// TIA Portal project "MOVE" (V19)

(* hardware
DEVICE "SIMATIC 1200 station_1"  S71200.Device
   slot 0: "S7-1200 rack"  Rack  V1.0
   slot 1: "PLC_1"  CPU 1214C DC/DC/DC  6ES7 214-1AG40-0XB0  V4.0
   slot 3: "AQ1 x 12 bits_1"  6ES7 232-4HA30-0XB0  V1.0
DEVICE "HMI_1"  KTP600 Basic color PN
   slot 0: "HMI"  HMI  6AV6 647-0AD11-3AX0  12.0.0.0
   slot 1: "HMI_RT_1"  KTP600 Basic color PN  6AV6 647-0AD11-3AX0  12.0.0.0
   slot 5: "IE_CP_1"  PROFINET Interface  IE_CP  V7.1.0
      slot 1: "PROFINET_Interface_1"  PROFINET Interface
         slot 1: "PORT_1"  Port  1.0.0.0
*)

// ===== PLC "PLC_1"  CPU 1214C DC/DC/DC =====

VAR_GLOBAL   // PLC tag table "Default tag table"
   "SEL_SW_1" AT %I0.0 : Bool;   // Selector Switch, Position 1
   "SEL_SW_2" AT %I0.1 : Bool;   // Selector Switch, Position 2
   "SEL_SW_3" AT %I0.2 : Bool;   // Selector Switch, Position 3
   "START" AT %I0.4 : Bool;   // START Momentary N. O. Pushbutton
   "OUTPUT" AT %Q0.0 : Bool;   // Process Output
END_VAR

DATA_BLOCK "Data_block_Presets"   // DB1
{ S7_Optimized_Access := 'TRUE' }
VERSION : 0.1
   VAR RETAIN
      PRE_SET_1 : Int := 10000;   // Preset No. 1
      PRE_SET_2 : Int := 15000;   // Preset No. 2
      PRE_SET_3 : Int := 20000;   // Preset No. 3
   END_VAR
   VAR
      ONE_SHOT : Array[0..2] of Bool;   // One Shot Control
   END_VAR
BEGIN
END_DATA_BLOCK

// folder: System blocks/Program resources

DATA_BLOCK "DWELL"   // DB2
{ S7_Optimized_Access := 'TRUE' }
AUTHOR : Simatic
FAMILY : IEC
NAME : IEC_TMR
VERSION : 1.0
// stored: InstanceOfName IEC_TIMER
"IEC_TIMER"
BEGIN
END_DATA_BLOCK

// folder: (top level)

ORGANIZATION_BLOCK "Main"   // OB1, LAD, ProgramCycle
TITLE = "Main Program Sweep (Cycle)"
{ S7_Optimized_Access := 'TRUE' }
VERSION : 0.1
BEGIN

REGION Network 1
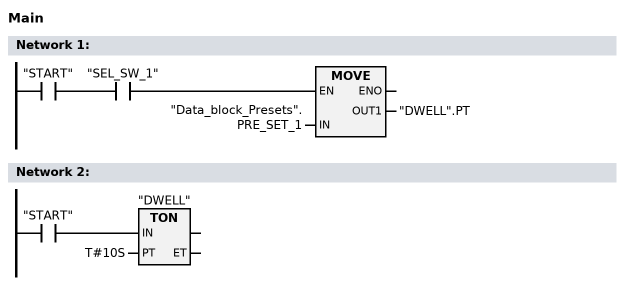
   RUNG wire#powerrail
      Contact( "START" )
      Contact( "SEL_SW_1" )
      Move(in := "Data_block_Presets".PRE_SET_1, out1 => "DWELL".PT)
   END_RUNG
   // the same network as SCL:
   IF "START" AND "SEL_SW_1" THEN "DWELL".PT := "Data_block_Presets".PRE_SET_1; END_IF;
END_REGION

REGION Network 2
   "DWELL".TON(IN := "START", PT := T#10S);
END_REGION
END_ORGANIZATION_BLOCK

(* ===== HMI "HMI_RT_1" =====
system functions are stored by id; their names below are inferred from use
connection "HMI_connection": ETHERNET, SMART_S7_1200_OMS

HMI tags "Default tag table"
   "OUTPUT" : Bool = PLC OUTPUT AT %Q0.0, 1 s
   "Data_block_HMI_OP_PB" : Int = PLC Data_block_HMI.HMI_PB, 1 s
   "Data_block_HMI_OP_START" : Bool = PLC Data_block_HMI.HMI_START, 1 s
   "Data_block_HMI_OP_PT" : Real = PLC Data_block_HMI.HMI_PT, 1 s
   "Data_block_HMI_OP_ET" : Real = PLC Data_block_HMI.HMI_ET, 1 s
   "Data_block_HMI_ENABLE_DISABLE" : Bool = PLC Data_block_HMI.HMI_ENABLE_DISABLE, 1 s
   "Data_block_Presets_PRE_SET_1" : Int = PLC Data_block_Presets.PRE_SET_1, 1 s
   "Data_block_Presets_PRE_SET_2" : Int = PLC Data_block_Presets.PRE_SET_2, 1 s
   "Data_block_Presets_PRE_SET_3" : Int = PLC Data_block_Presets.PRE_SET_3, 1 s

Template "Template_1" 320x240
   Softkey "Softkey_F6" at 266,202 size 53x38
      on KeyUp: StopRuntime(0)
   Button "Template_Button_1" at 268,202 size 51x37; TextOff 'Text'; PictureOff "ExitRuntime_HMI_1"
      on Release: StopRuntime(0)

screen "Root screen" 320x240, template "Template_1"
   GraphicView "D3_Plate_Vertical_Broad" at 13,33 size 106x165; Picture "Design_3_Plate_Vertical_Broad"
   GraphicView "D3_Plate_Vertical_Broad_1" at 128,33 size 184x164; Picture "Design_3_Plate_Vertical_Broad"
   Button "Button_1" at 47,60 size 36x36; TextOff '1'
      on Release: SetTag("Data_block_HMI_OP_PB", 1)
   TextField "Text field_1" at 25,38 size 80x18; Text 'TIME SELECT'
   Button "Button_2" at 47,104 size 36x36; TextOff '2'
      on Release: SetTag("Data_block_HMI_OP_PB", 2)
   Button "Button_3" at 47,149 size 36x36; TextOff '3'
      on Release: SetTag("Data_block_HMI_OP_PB", 3)
   IOField "I/O field_1" at 214,149 size 80x23; FormatPattern 99.99
      ProcessValue <- "Data_block_HMI_OP_ET"
   Button "Button_4" at 144,53 size 91x30; TextOff 'START'
      on Press: SetBit("Data_block_HMI_OP_START")
      on Release: ResetBit("Data_block_HMI_OP_START")
   IOField "I/O field_2" at 214,108 size 80x23; FormatPattern 99.99
      ProcessValue <- "Data_block_HMI_OP_PT"
   TextField "Text field_2" at 34,4 size 252x21; Text 'MOVE LAB OPERATORS PANEL'
   Circle "Circle_1" at 254,57 size 32x32
      Appearance <- "OUTPUT"
   TextField "Text field_4" at 140,106 size 68x15; Text 'TIME DELAY'
   TextField "Text field_5" at 150,117 size 48x16; Text 'PRESET'
   TextField "Text field_6" at 148,145 size 53x15; Text 'CURRENT'
   TextField "Text field_7" at 159,156 size 30x15; Text 'TIME'
   TextField "Text field_3" at 247,40 size 47x15; Text 'OUTPUT'
   Button "Button_5" at 1,202 size 51x37; TextOff 'SCREEN 2'
      on Release: ActivateScreen("Screen_2", 0)
   TextField "Text field_8" at 68,200 size 105x35; Text 'OVERRIDE FOR HARDWIRED OPERATOR'S PANEL'
   Switch "Switch_1" at 180,202 size 69x33; CaptionText 'Switch'; TextOff 'HMI DISABLED'; TextOn 'HMI ENABLED'
      ProcessValue <- "Data_block_HMI_ENABLE_DISABLE"
   Softkey "Softkey_F1" at 1,202 size 53x38
      on KeyUp: ActivateScreen("Screen_2", 0)

screen "Screen_2" 320x240, template "Template_1"
   Softkey "Softkey_F1" at 1,202 size 53x38
      on KeyUp: ActivateScreen("Root screen", 0)
   Button "Button_1" at 2,201 size 51x37; TextOff 'SCREEN 1'
      on Release: ActivateScreen("Root screen", 0)
   TextField "Text field_2" at 31,4 size 258x21; Text 'PRESET MAINTENANCE PANEL'
   GraphicView "D3_Plate_Vertical_Broad_1" at 59,34 size 203x163; Picture "Design_3_Plate_Vertical_Broad"
   TextField "Text field_1" at 81,41 size 160x28; Text 'ENTER VALUES AS INTEGERS TIMEBASE OF MILLISECONDS'
   TextField "Text field_3" at 82,77 size 60x18; Text 'PRESET 1'
   TextField "Text field_4" at 82,117 size 60x18; Text 'PRESET 2'
   TextField "Text field_5" at 82,158 size 60x18; Text 'PRESET 3'
   IOField "I/O field_1" at 155,73 size 74x26; FormatPattern 99999
      ProcessValue <- "Data_block_Presets_PRE_SET_1"
   IOField "I/O field_2" at 155,113 size 74x26; FormatPattern 99999
      ProcessValue <- "Data_block_Presets_PRE_SET_2"
   IOField "I/O field_3" at 155,153 size 74x26; FormatPattern 99999
      ProcessValue <- "Data_block_Presets_PRE_SET_3"
*)